VAR_GLOBAL
  PumpAlpha : FB_Device;
  FlowValue : REAL;
  ValveCommand : BOOL := FALSE;
END_VAR
